PROGRAM Sinalizadores
VAR
END_VAR

(*=================		SINALIZADORES LUMINOSOS		======================*)	

//Comando Ligado
IF (TRUE) THEN
	OutSinalizadorComandoLigado := TRUE;
ELSE
	OutSinalizadorComandoLigado := FALSE;
END_IF

//Botoeira HS1
IF (TRUE) THEN
	OutSinalizadorBotoeiraHS1 := TRUE;
ELSE
	OutSinalizadorBotoeiraHS1 := FALSE;
END_IF

//Botoeira HS2
IF (TRUE) THEN
	OutSinalizadorBotoeiraHS2 := TRUE;
ELSE
	OutSinalizadorBotoeiraHS2 := FALSE;
END_IF

(*========================================================================*)

END_PROGRAM

(* stored: Version 1.1.0.1, ProductVersion 3.1.4024.11
   POU Sinalizadores: Id {1137fa02-b690-41e0-825d-52a952bb0634}, SpecialFunc None *)
